FUNCTION Convert_BOOL_TO_UDINT : BOOL
VAR_INPUT
	in : BOOL;
	out : REFERENCE TO UDINT;
END_VAR

out := BOOL_TO_UDINT(in);
Convert_BOOL_TO_UDINT := TRUE;

END_FUNCTION

(* stored: Version 1.1.0.1, ProductVersion 3.1.4024.12
   POU Convert_BOOL_TO_UDINT: Id {2b512001-2e03-453e-8150-371a1c253f4b}, SpecialFunc None *)
